// SIMATIC S7-200 project (STEP 7-Micro/WIN), CPU 224XP CN REL 02.01

ORGANIZATION_BLOCK MAIN:OB1
TITLE=
BEGIN
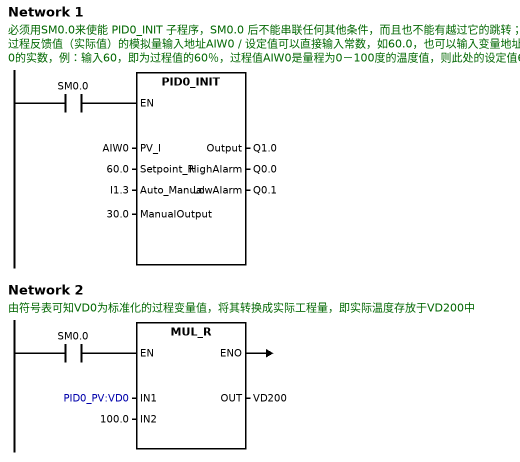
Network 1
// 必须用SM0.0来使能 PID0_INIT 子程序，SM0.0 后不能串联任何其他条件，而且也不能有越过它的跳转；如果在子程序中调用 PID0_INIT 子程序，则调用它的子程序也必须仅使用 SM0.0 调用，以保证它的正常运行
// 过程反馈值（实际值）的模拟量输入地址AIW0
// 设定值可以直接输入常数，如60.0，也可以输入变量地址（VDxx），根据向导中的设定0.0-100.0，此处应输入一个0.0－100.0的实数，例：输入60，即为过程值的60％，过程值AIW0是量程为0－100度的温度值，则此处的设定值60代表60度（即100度的60％）
// I1.3控制PID的手/自动方式，当I1.3为1时，为自动，经过PID运算从Q1.0输出；当I1.3为0时，PID将停止计算，Q1.0将输出为占空比30.0%的信号。若在向导中没有选择PID手动功能，则此项不会出现
// 30.0即为PID手动状态下的输出，此处可输入手动设定值的变量地址（VDxx），或直接输入常数。若在向导中没有选择PID手动功能，则此项不会出现
// 组态PID指令向导时，设置控制量的输出为数字量，此处Q1.0连接了一个加热器
// 当高限报警条件满足时，相应的输出置位为1，此处为Q0.0，若在向导中没有使能高限报警功能，则此项将不会出现
// 当低限报警条件满足时，相应的输出置位为1，此处为Q0.1，若在向导中没有使能低限报警功能，则此项将不会出现
// 当模块出错时，相应的输出置位为1，若在向导中没有使能模块错误报警功能，则此项将不会出现 
// (network saved uncompiled; LAD cells follow)
// row 0: c0 -| |- SM0.0  c1 [PID0_INIT EN:=power@row0, PV_I:=AIW0, Setpoint_R:=60.0, Auto_Manual:=I1.3, ManualOutput:=30.0, Output=>Q1.0, HighAlarm=>Q0.0, LowAlarm=>Q0.1]
// row 1: c1 [box]
// row 2: c1 [box]
Network 2
// 由符号表可知VD0为标准化的过程变量值，将其转换成实际工程量，即实际温度存放于VD200中
// (network saved uncompiled; LAD cells follow)
// row 0: c0 -| |- SM0.0  c1 [MUL_R EN:=power@row0, IN1:=PID0_PV:VD0, IN2:=100.0, ENO=>power, OUT=>VD200]  c2 ->
// row 1: c1 [box]
END_ORGANIZATION_BLOCK

// SBR1: protected block, not included

// INT1: protected block, not included

// (further data pages could not be read)
